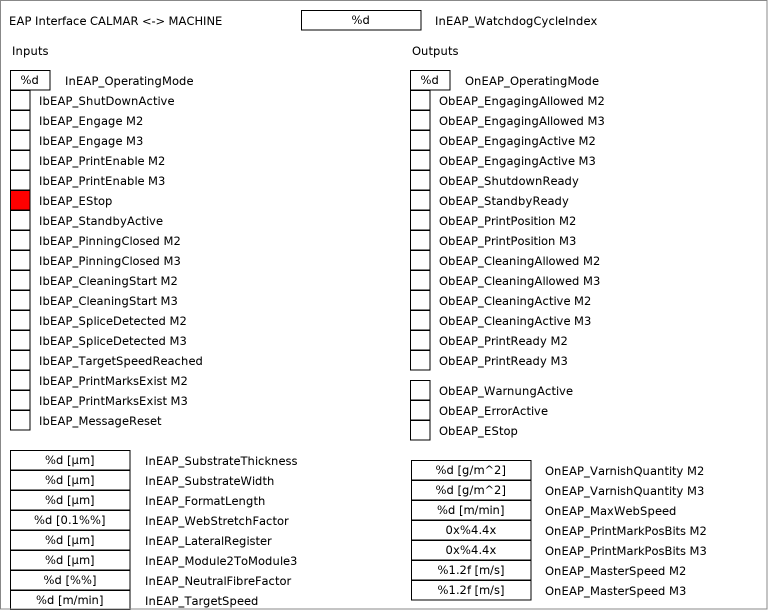
VISUALIZATION VISU_EAP_MACHINE  // 768x610
    RoundedRectangle (10,90 20x20), colour toggle: PRG_MACHINE.IbEAP_ShutDownActive
    RoundedRectangle (10,110 20x20), colour toggle: PRG_MACHINE.IbEAP_Engaged[1]
    RoundedRectangle (10,150 20x20), colour toggle: PRG_MACHINE.IbEAP_PrintEnabled[1]
    Rectangle (36,92 257x18), "IbEAP_ShutDownActive"
    Rectangle (36,112 256x18), "IbEAP_Engage M2"
    Rectangle (36,152 226x18), "IbEAP_PrintEnable M2"
    RoundedRectangle (10,190 20x20), colour toggle: NOT PRG_MACHINE.IbEAP_EStop
    Rectangle (36,192 226x18), "IbEAP_EStop"
    RoundedRectangle (10,210 20x20), colour toggle: PRG_MACHINE.IbEAP_StandbyActive
    Rectangle (36,212 226x18), "IbEAP_StandbyActive"
    RoundedRectangle (10,410 20x20), colour toggle: PRG_MACHINE.IbEAP_MessageReset
    Rectangle (36,412 226x18), "IbEAP_MessageReset"
    RoundedRectangle (10,230 20x20), colour toggle: PRG_MACHINE.IbEAP_PinningClosed[1]
    Rectangle (36,232 226x18), "IbEAP_PinningClosed M2"
    Rectangle (10,530 120x20), "%d [µm]", text variable: PRG_MACHINE.InEAP_LateralRegister
    Rectangle (142,532 226x18), "InEAP_LateralRegister"
    Rectangle (10,450 120x20), "%d [µm]", text variable: PRG_MACHINE.InEAP_SubstrateThickness
    Rectangle (142,452 226x18), "InEAP_SubstrateThickness"
    Rectangle (10,470 120x20), "%d [µm]", text variable: PRG_MACHINE.InEAP_SubstrateWidth
    Rectangle (142,472 226x18), "InEAP_SubstrateWidth"
    Rectangle (10,490 120x20), "%d [µm]", text variable: PRG_MACHINE.InEAP_FormatLength
    Rectangle (142,492 226x18), "InEAP_FormatLength"
    Rectangle (6,12 257x18), "EAP Interface CALMAR <-> MACHINE"
    RoundedRectangle (410,90 20x20), colour toggle: PRG_MACHINE.ObEAP_EngagingAllowed[1]
    Rectangle (436,92 257x18), "ObEAP_EngagingAllowed M2"
    RoundedRectangle (410,170 20x20), colour toggle: PRG_MACHINE.ObEAP_ShutdownReady
    Rectangle (436,172 257x18), "ObEAP_ShutdownReady"
    RoundedRectangle (410,190 20x20), colour toggle: PRG_MACHINE.ObEAP_StandbyReady
    Rectangle (436,192 257x18), "ObEAP_StandbyReady"
    RoundedRectangle (410,210 20x20), colour toggle: PRG_MACHINE.ObEAP_PrintPosition[1]
    Rectangle (436,212 257x18), "ObEAP_PrintPosition M2"
    Rectangle (9,42 257x18), "Inputs"
    Rectangle (409,42 257x18), "Outputs"
    Rectangle (411,480 120x20), "%d [g/m^2]", text variable: PRG_MACHINE.OnEAP_VarnishQuantity[2]
    Rectangle (542,482 226x18), "OnEAP_VarnishQuantity M3"
    Rectangle (411,500 120x20), "%d [m/min]", text variable: PRG_MACHINE.OnEAP_MaxWebSpeed
    Rectangle (542,502 226x18), "OnEAP_MaxWebSpeed"
    Rectangle (301,10 120x20), "%d", text variable: PRG_MACHINE.InEAP_WatchdogCycleIndex
    Rectangle (432,12 226x18), "InEAP_WatchdogCycleIndex"
    RoundedRectangle (410,380 20x20), colour toggle: PRG_MACHINE.ObEAP_WarnungActive
    Rectangle (436,382 257x18), "ObEAP_WarnungActive"
    RoundedRectangle (410,400 20x20), colour toggle: PRG_MACHINE.ObEAP_ErrorActive
    Rectangle (436,402 257x18), "ObEAP_ErrorActive"
    RoundedRectangle (10,270 20x20), colour toggle: PRG_MACHINE.IbEAP_CleaningStart[1]
    Rectangle (36,272 226x18), "IbEAP_CleaningStart M2"
    RoundedRectangle (410,250 20x20), colour toggle: PRG_MACHINE.ObEAP_CleaningAllowed[1]
    Rectangle (436,252 257x18), "ObEAP_CleaningAllowed M2"
    RoundedRectangle (410,310 20x20), colour toggle: PRG_MACHINE.ObEAP_CleaningActive[2]
    Rectangle (436,312 257x18), "ObEAP_CleaningActive M3"
    RoundedRectangle (410,330 20x20), colour toggle: PRG_MACHINE.ObEAP_PrintReady[1]
    Rectangle (436,332 257x18), "ObEAP_PrintReady M2"
    Rectangle (10,510 120x20), "%d [0.1%%]", text variable: PRG_MACHINE.InEAP_WebStretchFactor
    Rectangle (142,512 226x18), "InEAP_WebStretchFactor"
    Rectangle (410,70 40x20), "%d", text variable: PRG_MACHINE.OnEAP_OperatingMode
    Rectangle (462,72 171x18), "OnEAP_OperatingMode"
    Rectangle (10,70 40x20), "%d", text variable: PRG_MACHINE.InEAP_OperatingMode
    Rectangle (62,72 171x18), "InEAP_OperatingMode"
    RoundedRectangle (10,130 20x20), colour toggle: PRG_MACHINE.IbEAP_Engaged[2]
    Rectangle (36,132 256x18), "IbEAP_Engage M3"
    RoundedRectangle (10,170 20x20), colour toggle: PRG_MACHINE.IbEAP_PrintEnabled[2]
    Rectangle (36,172 226x18), "IbEAP_PrintEnable M3"
    RoundedRectangle (10,290 20x20), colour toggle: PRG_MACHINE.IbEAP_CleaningStart[2]
    Rectangle (36,292 226x18), "IbEAP_CleaningStart M3"
    RoundedRectangle (10,250 20x20), colour toggle: PRG_MACHINE.IbEAP_PinningClosed[2]
    Rectangle (36,252 226x18), "IbEAP_PinningClosed M3"
    RoundedRectangle (410,110 20x20), colour toggle: PRG_MACHINE.ObEAP_EngagingAllowed[2]
    Rectangle (436,112 257x18), "ObEAP_EngagingAllowed M3"
    RoundedRectangle (410,130 20x20), colour toggle: PRG_MACHINE.ObEAP_EngagingActive[1]
    Rectangle (436,132 257x18), "ObEAP_EngagingActive M2"
    RoundedRectangle (410,150 20x20), colour toggle: PRG_MACHINE.ObEAP_EngagingActive[2]
    Rectangle (436,152 257x18), "ObEAP_EngagingActive M3"
    RoundedRectangle (410,230 20x20), colour toggle: PRG_MACHINE.ObEAP_PrintPosition[2]
    Rectangle (436,232 257x18), "ObEAP_PrintPosition M3"
    RoundedRectangle (410,270 20x20), colour toggle: PRG_MACHINE.ObEAP_CleaningAllowed[2]
    Rectangle (436,272 257x18), "ObEAP_CleaningAllowed M3"
    RoundedRectangle (410,290 20x20), colour toggle: PRG_MACHINE.ObEAP_CleaningActive[1]
    Rectangle (436,292 257x18), "ObEAP_CleaningActive M2"
    RoundedRectangle (410,350 20x20), colour toggle: PRG_MACHINE.ObEAP_PrintReady[2]
    Rectangle (436,352 257x18), "ObEAP_PrintReady M3"
    Rectangle (411,460 120x20), "%d [g/m^2]", text variable: PRG_MACHINE.OnEAP_VarnishQuantity[1]
    Rectangle (542,462 226x18), "OnEAP_VarnishQuantity M2"
    RoundedRectangle (10,310 20x20), colour toggle: PRG_MACHINE.IbEAP_SpliceDetected[1]
    Rectangle (36,312 226x18), "IbEAP_SpliceDetected M2"
    RoundedRectangle (10,330 20x20), colour toggle: PRG_MACHINE.IbEAP_SpliceDetected[2]
    Rectangle (36,332 226x18), "IbEAP_SpliceDetected M3"
    Rectangle (10,550 120x20), "%d [µm]", text variable: PRG_MACHINE.InEAP_Module2ToModule3
    Rectangle (142,552 226x18), "InEAP_Module2ToModule3"
    RoundedRectangle (10,350 20x20), colour toggle: PRG_MACHINE.IbEAP_TargetSpeedReached]
    Rectangle (36,352 226x18), "IbEAP_TargetSpeedReached"
    RoundedRectangle (10,370 20x20), colour toggle: PRG_MACHINE.IbEAP_PrintMarksExist[1]
    Rectangle (36,372 226x18), "IbEAP_PrintMarksExist M2"
    RoundedRectangle (10,390 20x20), colour toggle: PRG_MACHINE.IbEAP_PrintMarksExist[2]
    Rectangle (36,392 226x18), "IbEAP_PrintMarksExist M3"
    Rectangle (10,570 120x20), "%d [%%]", text variable: PRG_MACHINE.InEAP_NeutralFibreFactor
    Rectangle (142,572 226x18), "InEAP_NeutralFibreFactor"
    Rectangle (10,590 120x20), "%d [m/min]", text variable: PRG_MACHINE.InEAP_NeutralFibreFactor
    Rectangle (142,592 226x18), "InEAP_TargetSpeed"
    RoundedRectangle (410,420 20x20), colour toggle: PRG_MACHINE.ObEAP_ErrorActive
    Rectangle (436,422 257x18), "ObEAP_EStop"
    Rectangle (411,540 120x20), "0x%4.4x", text variable: PRG_MACHINE.OnEAP_PrintMarkPosBits[2]
    Rectangle (542,542 226x18), "OnEAP_PrintMarkPosBits M3"
    Rectangle (411,520 120x20), "0x%4.4x", text variable: PRG_MACHINE.OnEAP_PrintMarkPosBits[1]
    Rectangle (542,522 226x18), "OnEAP_PrintMarkPosBits M2"
    Rectangle (411,580 120x20), "%1.2f [m/s]", text variable: PRG_MACHINE.OnEAP_MasterSpeed[2]
    Rectangle (542,582 226x18), "OnEAP_MasterSpeed M3"
    Rectangle (411,560 120x20), "%1.2f [m/s]", text variable: PRG_MACHINE.OnEAP_MasterSpeed[1]
    Rectangle (542,562 226x18), "OnEAP_MasterSpeed M2"
END_VISUALIZATION

(* stored: Version 1.1.0.1, ProductVersion 3.1.4024.9
   Visu VISU_EAP_MACHINE: Id {24a16f96-388e-425e-afbb-8aa4100e25d0} *)
